// TIA Portal project "Napelnianie_zbiornika" (V15.1)

(* hardware
DEVICE "S71500/ET200MP station_1"  S7-1500 station
   slot 0: "Rail_0"  Rack  6ES7 590-1***0-0AA0
   slot 1: "PLC_3"  CPU 1511TF-1 PN  6ES7 511-1UK01-0AB0  V2.6
      slot 3: "CPU display_1"  6ES7591-1AA00-0AA0
*)

// ===== PLC "PLC_3"  CPU 1511TF-1 PN =====

VAR_GLOBAL   // PLC tag table "Default tag table"
   "System_Byte" AT %MB1000 : Byte;
   "FirstScan" AT %M1000.0 : Bool;
   "DiagStatusUpdate" AT %M1000.1 : Bool;
   "AlwaysTRUE" AT %M1000.2 : Bool;
   "AlwaysFALSE" AT %M1000.3 : Bool;
   "System_Byte(1)" AT %MB1 : Byte;
   "Clock_Byte" AT %MB1010 : Byte;
   "Clock_10Hz" AT %M1010.0 : Bool;
   "Clock_5Hz" AT %M1010.1 : Bool;
   "Clock_2.5Hz" AT %M1010.2 : Bool;
   "Clock_2Hz" AT %M1010.3 : Bool;
   "Clock_1.25Hz" AT %M1010.4 : Bool;
   "Clock_1Hz" AT %M1010.5 : Bool;
   "Clock_0.625Hz" AT %M1010.6 : Bool;
   "Clock_0.5Hz" AT %M1010.7 : Bool;
END_VAR

DATA_BLOCK "Dane_funkcji"   // DB1
{ S7_Optimized_Access := 'TRUE' }
VERSION : 0.1
// stored: InstanceOfName Zbiornik
"Zbiornik"
BEGIN
END_DATA_BLOCK

DATA_BLOCK "Blok danych"   // DB3
{ S7_Optimized_Access := 'TRUE' }
VERSION : 0.1
   VAR
      start : Bool;
      "predkosc_oprozniania[m3/s]" : Real := 1.0;
      stop : Bool;
      napelnianie : Bool;
      oproznianie : Bool;
      zalacz : Bool;
      napelnij : Bool;
      oproznij : Bool;
      "objetosc[litry]" : Real;
      "stan alarmowy" : Bool;
      "pojemnosc[ml]" : ULInt := 10000000;
      przepelnienie : Bool;
      "predkosc_napelniania[m3/s]" : Real := 1.0;
      Impulsy : Bool;
      "zb. narast" : Bool;
      "zb. opad" : Bool;
      "generator 1HZ" : Bool;
      "Wysokosc [m]" : Real;
   END_VAR
BEGIN
END_DATA_BLOCK

FUNCTION_BLOCK "Zbiornik"   // FB1, LAD
{ S7_Optimized_Access := 'TRUE' }
VERSION : 0.1
   VAR_INPUT
      pr_napelniania : Real := 0.0;
      pr_oprozniania : Real;
      Pojemnosc : Real;
      Napelnianie : Bool;
      Oproznianie : Bool;
   END_VAR
   VAR_OUTPUT
      Aktualna_objetosc : Real;
      Stan_alarmowy : Bool;
      "Poziom cieczyy" : Real;
      "Przepelnienie_100%" : Bool;
   END_VAR
   VAR
      kontrola : Bool;
      kontrola_1 : Bool;
      "Przepelnienie_120%" : Real;
      "Alarm_85%" : Real;
      "Przyrost obj" : Real;
      "Spadek obj" : Real;
      "Alarm_100%" : Real;
   END_VAR
   VAR CONSTANT
      Alarm_85 : Real := 0.00085;
      Alarm_120 : Real := 0.0012;
      Predkosc_min : Real := 0.0;
      Predkosc_max : Real := 1.0;
      "Powierzchnia [dm2]" : Real := 2998.4;
      Minimum : Int;
      Alarm_100 : Real := 0.001;
   END_VAR
   VAR_TEMP   // added for the SCL form of the ladder/FBD networks
      _w1 : Bool;
      _w2 : Bool;
   END_VAR
BEGIN

REGION Network 1: Generowanie zbocza+ograniczenie predkosci
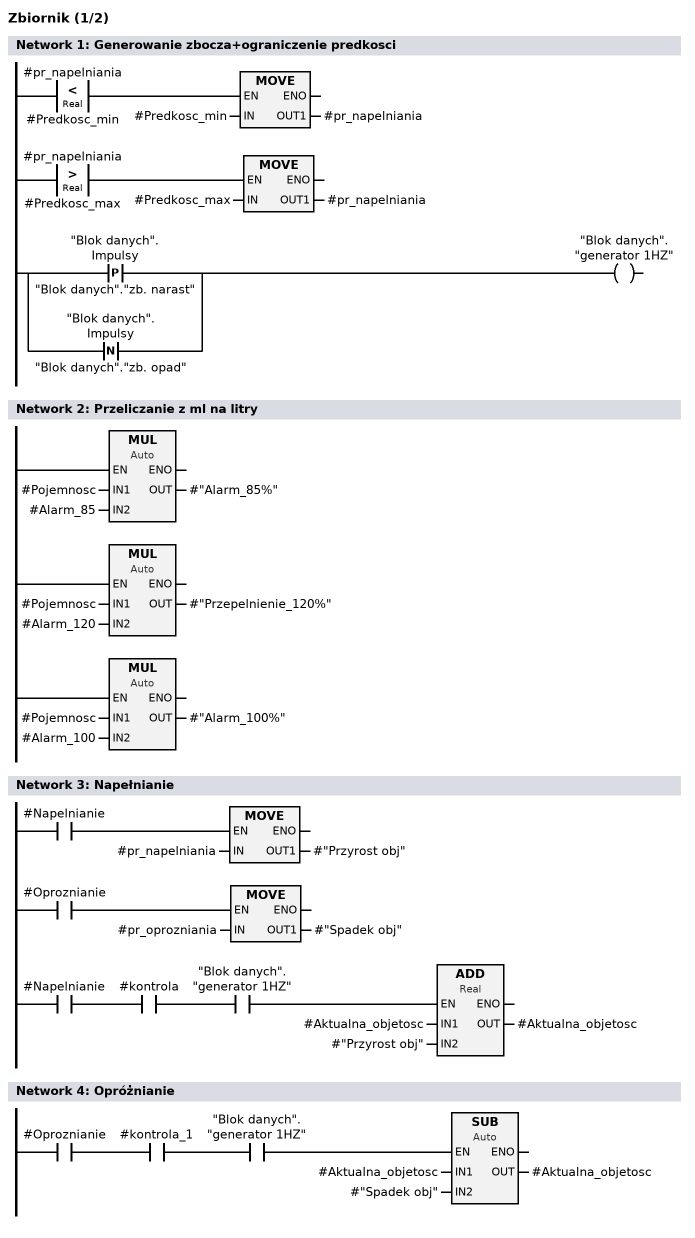
   RUNG wire#powerrail
      { S7_Templates := "SrcType := Real" } LT_Contact(in1 := #pr_napelniania, in2 := #Predkosc_min)
      Move(in := #Predkosc_min, out1 => #pr_napelniania)
   END_RUNG
   RUNG wire#powerrail
      { S7_Templates := "SrcType := Real" } GT_Contact(in1 := #pr_napelniania, in2 := #Predkosc_max)
      Move(in := #Predkosc_max, out1 => #pr_napelniania)
   END_RUNG
   RUNG wire#powerrail
      P_Contact(operand := "Blok danych".Impulsy, bit := "Blok danych"."zb. narast")
      wire#w1
      Coil( "Blok danych"."generator 1HZ" )
   END_RUNG
   RUNG wire#powerrail
      N_Contact(operand := "Blok danych".Impulsy, bit := "Blok danych"."zb. opad")
   END_RUNG wire#w1
   // the same network as SCL:
   IF #pr_napelniania < #Predkosc_min THEN #pr_napelniania := #Predkosc_min; END_IF;
   IF #pr_napelniania > #Predkosc_max THEN #pr_napelniania := #Predkosc_max; END_IF;
   #_w1 := "Blok danych".Impulsy AND NOT "Blok danych"."zb. narast";   // rising edge of "Blok danych".Impulsy
   "Blok danych"."zb. narast" := "Blok danych".Impulsy;
   #_w2 := NOT "Blok danych".Impulsy AND "Blok danych"."zb. opad";   // falling edge of "Blok danych".Impulsy
   "Blok danych"."zb. opad" := "Blok danych".Impulsy;
   "Blok danych"."generator 1HZ" := #_w1 OR #_w2;
END_REGION

REGION Network 2: Przeliczanie z ml na litry
   RUNG wire#powerrail
      Mul(in1 := #Pojemnosc, in2 := #Alarm_85, out => #"Alarm_85%")
   END_RUNG
   RUNG wire#powerrail
      Mul(in1 := #Pojemnosc, in2 := #Alarm_120, out => #"Przepelnienie_120%")
   END_RUNG
   RUNG wire#powerrail
      Mul(in1 := #Pojemnosc, in2 := #Alarm_100, out => #"Alarm_100%")
   END_RUNG
   // the same network as SCL:
   #"Alarm_85%" := #Pojemnosc * #Alarm_85;
   #"Przepelnienie_120%" := #Pojemnosc * #Alarm_120;
   #"Alarm_100%" := #Pojemnosc * #Alarm_100;
END_REGION

REGION Network 3: Napełnianie
   RUNG wire#powerrail
      Contact( #Napelnianie )
      Move(in := #pr_napelniania, out1 => #"Przyrost obj")
   END_RUNG
   RUNG wire#powerrail
      Contact( #Oproznianie )
      Move(in := #pr_oprozniania, out1 => #"Spadek obj")
   END_RUNG
   RUNG wire#powerrail
      Contact( #Napelnianie )
      Contact( #kontrola )
      Contact( "Blok danych"."generator 1HZ" )
      { S7_Templates := "SrcType := Real" } Add(in1 := #Aktualna_objetosc, in2 := #"Przyrost obj", out => #Aktualna_objetosc)
   END_RUNG
   // the same network as SCL:
   IF #Napelnianie THEN #"Przyrost obj" := #pr_napelniania; END_IF;
   IF #Oproznianie THEN #"Spadek obj" := #pr_oprozniania; END_IF;
   IF #Napelnianie AND #kontrola AND "Blok danych"."generator 1HZ" THEN
       #Aktualna_objetosc := #Aktualna_objetosc + #"Przyrost obj";
   END_IF;
END_REGION

REGION Network 4: Opróżnianie
   RUNG wire#powerrail
      Contact( #Oproznianie )
      Contact( #kontrola_1 )
      Contact( "Blok danych"."generator 1HZ" )
      Sub(in1 := #Aktualna_objetosc, in2 := #"Spadek obj", out => #Aktualna_objetosc)
   END_RUNG
   // the same network as SCL:
   IF #Oproznianie AND #kontrola_1 AND "Blok danych"."generator 1HZ" THEN
       #Aktualna_objetosc := #Aktualna_objetosc - #"Spadek obj";
   END_IF;
END_REGION

REGION Network 5: Alarmy
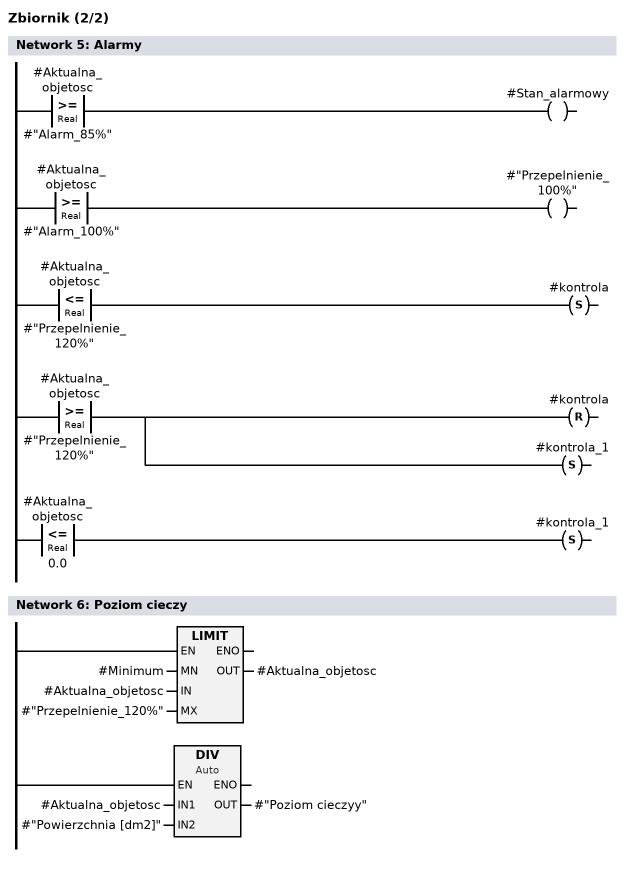
   RUNG wire#powerrail
      { S7_Templates := "SrcType := Real" } GE_Contact(in1 := #Aktualna_objetosc, in2 := #"Alarm_85%")
      Coil( #Stan_alarmowy )
   END_RUNG
   RUNG wire#powerrail
      { S7_Templates := "SrcType := Real" } GE_Contact(in1 := #Aktualna_objetosc, in2 := #"Alarm_100%")
      Coil( #"Przepelnienie_100%" )
   END_RUNG
   RUNG wire#powerrail
      { S7_Templates := "SrcType := Real" } LE_Contact(in1 := #Aktualna_objetosc, in2 := #"Przepelnienie_120%")
      S_Coil( #kontrola )
   END_RUNG
   RUNG wire#powerrail
      { S7_Templates := "SrcType := Real" } GE_Contact(in1 := #Aktualna_objetosc, in2 := #"Przepelnienie_120%")
      wire#w1
      R_Coil( #kontrola )
   END_RUNG
   RUNG wire#w1
      S_Coil( #kontrola_1 )
   END_RUNG
   RUNG wire#powerrail
      { S7_Templates := "SrcType := Real" } LE_Contact(in1 := #Aktualna_objetosc, in2 := 0.0)
      S_Coil( #kontrola_1 )
   END_RUNG
   // the same network as SCL:
   #Stan_alarmowy := #Aktualna_objetosc >= #"Alarm_85%";
   #"Przepelnienie_100%" := #Aktualna_objetosc >= #"Alarm_100%";
   IF #Aktualna_objetosc <= #"Przepelnienie_120%" THEN #kontrola := TRUE; END_IF;
   IF #Aktualna_objetosc >= #"Przepelnienie_120%" THEN
       #kontrola := FALSE;
       #kontrola_1 := TRUE;
   END_IF;
   IF #Aktualna_objetosc <= 0.0 THEN #kontrola_1 := TRUE; END_IF;
END_REGION

REGION Network 6: Poziom cieczy
   #Aktualna_objetosc := LIMIT(MN := #Minimum, IN := #Aktualna_objetosc, MX := #"Przepelnienie_120%");
   #"Poziom cieczyy" := #Aktualna_objetosc / #"Powierzchnia [dm2]";
END_REGION
END_FUNCTION_BLOCK

ORGANIZATION_BLOCK "Main"   // OB1, LAD, ProgramCycle
TITLE = "Main Program Sweep (Cycle)"
{ S7_Optimized_Access := 'TRUE' }
VERSION : 0.1
   VAR_INPUT
      Initial_Call : Bool;   // Initial call of this OB
      Remanence : Bool;   // =True, if remanent data are available
   END_VAR
BEGIN

REGION Network 2
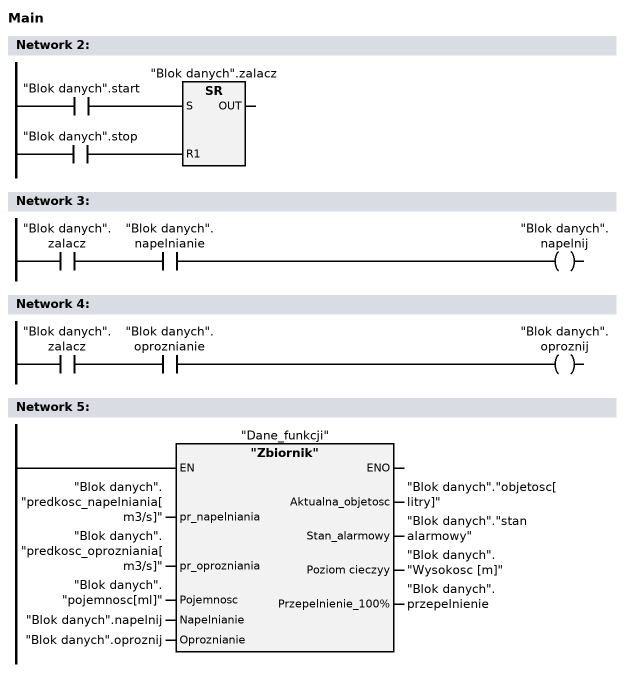
   RUNG wire#powerrail
      Contact( "Blok danych".start )
      S_SR(operand := "Blok danych".zalacz, r1 := wire#w1)
   END_RUNG
   RUNG wire#powerrail
      Contact( "Blok danych".stop )
   END_RUNG wire#w1
   // the same network as SCL:
   IF "Blok danych".start THEN
       "Blok danych".zalacz := TRUE;   // SR flip-flop
   END_IF;
   IF "Blok danych".stop THEN "Blok danych".zalacz := FALSE; END_IF;
END_REGION

REGION Network 3
   RUNG wire#powerrail
      Contact( "Blok danych".zalacz )
      Contact( "Blok danych".napelnianie )
      Coil( "Blok danych".napelnij )
   END_RUNG
   // the same network as SCL:
   "Blok danych".napelnij := "Blok danych".zalacz AND "Blok danych".napelnianie;
END_REGION

REGION Network 4
   RUNG wire#powerrail
      Contact( "Blok danych".zalacz )
      Contact( "Blok danych".oproznianie )
      Coil( "Blok danych".oproznij )
   END_RUNG
   // the same network as SCL:
   "Blok danych".oproznij := "Blok danych".zalacz AND "Blok danych".oproznianie;
END_REGION

REGION Network 5
   RUNG wire#powerrail
      "Dane_funkcji"(pr_napelniania := "Blok danych"."predkosc_napelniania[m3/s]", pr_oprozniania := "Blok danych"."predkosc_oprozniania[m3/s]", Pojemnosc := "Blok danych"."pojemnosc[ml]", Napelnianie := "Blok danych".napelnij, Oproznianie := "Blok danych".oproznij, Aktualna_objetosc => "Blok danych"."objetosc[litry]", Stan_alarmowy => "Blok danych"."stan alarmowy", "Poziom cieczyy" => "Blok danych"."Wysokosc [m]", "Przepelnienie_100%" => "Blok danych".przepelnienie)
   END_RUNG
   // the same network as SCL:
   "Dane_funkcji"(pr_napelniania := "Blok danych"."predkosc_napelniania[m3/s]",   // "Zbiornik"
                  pr_oprozniania := "Blok danych"."predkosc_oprozniania[m3/s]",
                  Pojemnosc := "Blok danych"."pojemnosc[ml]",
                  Napelnianie := "Blok danych".napelnij,
                  Oproznianie := "Blok danych".oproznij,
                  Aktualna_objetosc => "Blok danych"."objetosc[litry]",
                  Stan_alarmowy => "Blok danych"."stan alarmowy",
                  "Poziom cieczyy" => "Blok danych"."Wysokosc [m]",
                  "Przepelnienie_100%" => "Blok danych".przepelnienie);
END_REGION
END_ORGANIZATION_BLOCK

ORGANIZATION_BLOCK "Generator 1Hz"   // OB30, LAD, CyclicInterrupt
{ S7_Optimized_Access := 'TRUE' }
VERSION : 0.1
   VAR_INPUT
      Initial_Call : Bool;   // Initial call of this OB
      Event_Count : Int;   // Events discarded
   END_VAR
BEGIN

REGION Network 1
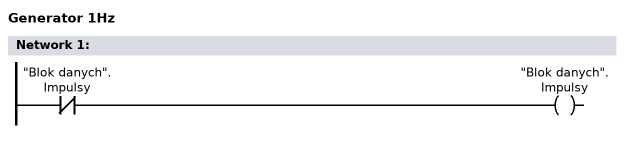
   RUNG wire#powerrail
      I_Contact( "Blok danych".Impulsy )
      Coil( "Blok danych".Impulsy )
   END_RUNG
   // the same network as SCL:
   "Blok danych".Impulsy := NOT "Blok danych".Impulsy;
END_REGION
END_ORGANIZATION_BLOCK